// TIA Portal V17 export
// export: Created 2021-12-03T08:08:00.5371119Z, ExportSetting WithDefaults, DisplayName Totally Integrated Automation Portal, DisplayVersion V17, DisplayName TIA Portal Openness, DisplayVersion V17, DisplayName TIA Portal Version Control Interface, DisplayVersion V17, DisplayName STEP 7 Professional, DisplayVersion V17, DisplayName STEP 7 Safety, DisplayVersion V17, DisplayName WinCC Advanced, DisplayVersion V17
VAR_GLOBAL   // PLC tag table "Clock_Memory"
   M_Clock_Byte AT %MB0 : Byte;
   M_Clock_10Hz AT %M0.0 : Bool;
   M_Clock_5Hz AT %M0.1 : Bool;
   "M_Clock_2.5Hz" AT %M0.2 : Bool;
   M_Clock_2Hz AT %M0.3 : Bool;
   "M_Clock_1.25Hz" AT %M0.4 : Bool;
   M_Clock_1Hz AT %M0.5 : Bool;
   "M_Clock_0.625Hz" AT %M0.6 : Bool;
   "M_Clock_0.5Hz" AT %M0.7 : Bool;
   Always_True AT %M1.0 : Bool;
   Always_False AT %M1.1 : Bool;
END_VAR
